// Mitsubishi GX Works2 project: WaterPump   PLC: FX3U/FX3UC

// global labels: Global1
VAR_GLOBAL
  Run AT M0 : BOOL;
  RunStop AT M1 : BOOL;
  ClockSet AT M8015 : BOOL;
  ClockYear AT D8018 : INT;
  ClockMonth AT D8017 : INT;
  ClockDay AT D8016 : INT;
  ClockHour AT D8015 : INT;
  ClockMinute AT D8014 : INT;
  ClockSecond AT D8013 : INT;
  RunI AT X000 : BOOL;
  RunStopI AT X001 : BOOL;
  EmptyI AT X002 : BOOL;
  Empty AT M2 : BOOL;
  PumpTimer AT TC0 : BOOL;
  PumpO AT Y005 : BOOL;
  PumpCount AT D2 : INT;
  RunState AT D0 : INT;
  Pump AT M3 : BOOL;
  PumpCycleActive AT M4 : BOOL;
  PumpTimerDelay AT D1 : INT;
  PumpTimeMinuteNext AT D3 : INT;
END_VAR

// task Task_01 (event TRUE, interval 0, priority 31): POU_01

PROGRAM POU_01
VAR
  fTmp : BOOL;
  fPumpTime : BOOL;
  fClockDayMinute : INT;
  fPumpTimerEN : BOOL;
  fHourFrom : INT;
  fHourTo : INT;
  fMinuteSpace : INT;
  fPumpActiveDelay : INT;
  fPumpPassiveDelay : INT;
  fTest : BOOL;
END_VAR
RST(M8002, RunState);
MOV(M8002, 22, fHourFrom);
MOV(M8002, 5, fHourTo);
MOV(M8002, 60 * 2, fMinuteSpace);
MOV(M8002, 600 * 20, fPumpActiveDelay);
MOV(M8002, 600 * 10, fPumpPassiveDelay);
RST(M8002, fTest);

SET(M8000 AND Run, fTmp);
RST(fTmp, Run);
MOV(fTmp, 1, RunState);
RST(fTmp, fTmp);
SET(M8000 AND RunStop, fTmp);
RST(fTmp, RunState);
RST(fTmp, Pump);
RST(fTmp, fTmp);

RST(FALSE, ClockSet);
RST(FALSE, ClockYear); RST(FALSE, ClockMonth); RST(FALSE, ClockDay);
RST(FALSE, ClockHour); RST(FALSE, ClockMinute); RST(FALSE, ClockSecond);

(*active pump*)
SET(RunState = 1, fTmp);
SET(fTmp, Pump);
MOV(fTmp, fPumpActiveDelay, PumpTimerDelay);
MOV(fTmp, 10, RunState);
RST(fTmp, fTmp);
(*passive pump*)
SET(RunState = 2, fTmp);
SET(fTmp, Pump);
MOV(fTmp, fPumpPassiveDelay, PumpTimerDelay);
MOV(fTmp, 10, RunState);
RST(fTmp, fTmp);
(*stop after delay or full*)
OUT(RunState = 10, fPumpTimerEN);
OUT_T(fPumpTimerEN, PumpTimer, PumpTimerDelay);
SET(fPumpTimerEN AND (PumpTimer OR NOT Empty), fTmp);
RST(fTmp, Pump);
RST(fTmp, RunState);
RST(fTmp, fTmp);

(*toggle, reset count when enable*)
OUT(ClockHour >= fHourFrom OR ClockHour <= fHourTo, fPumpTime);
SET(fPumpTime AND NOT PumpCycleActive, fTmp);
RST(fTmp, PumpCount);
RST(fTmp, PumpTimeMinuteNext);
SET(fTmp, PumpCycleActive);
RST(fTmp, fTmp);
RST(NOT fPumpTime AND PumpCycleActive, PumpCycleActive);
(*decide*)
MOV(M8000 AND ClockHour >= fHourFrom, ClockHour * 60 + ClockMinute, fClockDayMinute);
MOV(M8000 AND ClockHour <= fHourTo, (ClockHour + 24) * 60 + ClockMinute, fClockDayMinute);
SET(M8000 AND PumpCycleActive AND Empty AND PumpCount < 3 AND fClockDayMinute > PumpTimeMinuteNext, fTmp);
MOV(fTmp, fClockDayMinute + fMinuteSpace, PumpTimeMinuteNext);
MOV(fTmp, 2, RunState);
INC(fTmp, PumpCount);
RST(fTmp, fTmp);

SET(NOT fTest AND RunI, Run); RST(NOT fTest AND NOT RunI, Run);
SET(NOT fTest AND RunStopI, RunStop); RST(NOT fTest AND NOT RunStopI, RunStop);
SET(NOT fTest AND EmptyI, Empty); RST(NOT fTest AND NOT EmptyI, Empty);

OUT(Pump, PumpO);
END_PROGRAM
